// TIA Portal V20 export
FUNCTION "04 T10 LANT Transitions" : Void   // FC1493, LAD
TITLE = TRANSITIONS
{ S7_Optimized_Access := 'TRUE' }
// stored: AutoNumber false, SetENOAutomatically false
   VAR_TEMP
      Aux_real : Real;
   END_VAR
BEGIN

REGION Network 1: ============ TRANSITIONS ============
END_REGION

REGION Network 2: Transitions - Zone Status
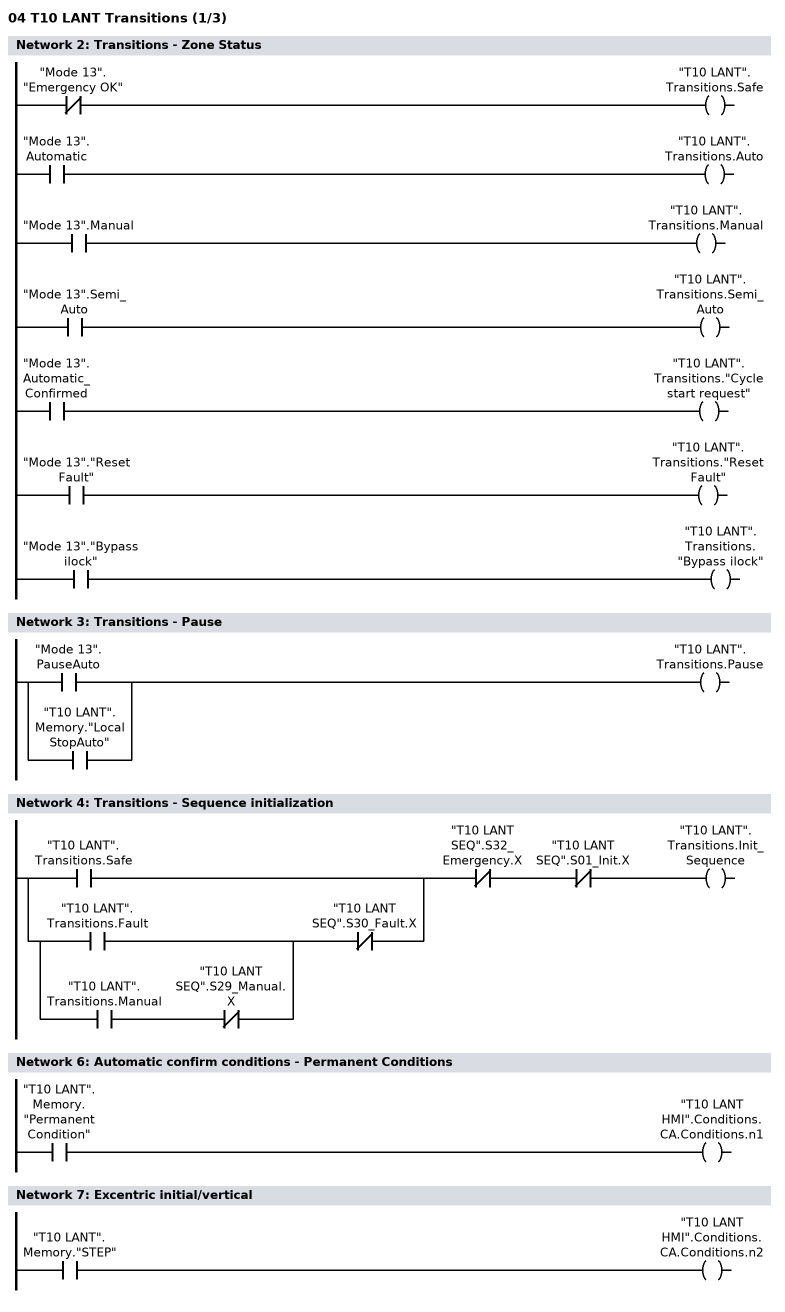
   RUNG wire#powerrail
      I_Contact( "Mode 13"."Emergency OK" )
      Coil( "T10 LANT".Transitions.Safe )
   END_RUNG
   RUNG wire#powerrail
      Contact( "Mode 13".Automatic )
      Coil( "T10 LANT".Transitions.Auto )
   END_RUNG
   RUNG wire#powerrail
      Contact( "Mode 13".Manual )
      Coil( "T10 LANT".Transitions.Manual )
   END_RUNG
   RUNG wire#powerrail
      Contact( "Mode 13".Semi_Auto )
      Coil( "T10 LANT".Transitions.Semi_Auto )
   END_RUNG
   RUNG wire#powerrail
      Contact( "Mode 13".Automatic_Confirmed )
      Coil( "T10 LANT".Transitions."Cycle start request" )
   END_RUNG
   RUNG wire#powerrail
      Contact( "Mode 13"."Reset Fault" )
      Coil( "T10 LANT".Transitions."Reset Fault" )
   END_RUNG
   RUNG wire#powerrail
      Contact( "Mode 13"."Bypass ilock" )
      Coil( "T10 LANT".Transitions."Bypass ilock" )
   END_RUNG
   // the same network as SCL:
   "T10 LANT".Transitions.Safe := NOT "Mode 13"."Emergency OK";
   "T10 LANT".Transitions.Auto := "Mode 13".Automatic;
   "T10 LANT".Transitions.Manual := "Mode 13".Manual;
   "T10 LANT".Transitions.Semi_Auto := "Mode 13".Semi_Auto;
   "T10 LANT".Transitions."Cycle start request" := "Mode 13".Automatic_Confirmed;
   "T10 LANT".Transitions."Reset Fault" := "Mode 13"."Reset Fault";
   "T10 LANT".Transitions."Bypass ilock" := "Mode 13"."Bypass ilock";
END_REGION

REGION Network 3: Transitions - Pause
   RUNG wire#powerrail
      Contact( "Mode 13".PauseAuto )
      wire#w1
      Coil( "T10 LANT".Transitions.Pause )
   END_RUNG
   RUNG wire#powerrail
      Contact( "T10 LANT".Memory."Local StopAuto" )
   END_RUNG wire#w1
   // the same network as SCL:
   "T10 LANT".Transitions.Pause := "Mode 13".PauseAuto OR "T10 LANT".Memory."Local StopAuto";
END_REGION

REGION Network 4: Transitions - Sequence initialization
   RUNG wire#powerrail
      Contact( "T10 LANT".Transitions.Safe )
      wire#w1
      I_Contact( "T10 LANT SEQ".S32_Emergency.X )
      I_Contact( "T10 LANT SEQ".S01_Init.X )
      Coil( "T10 LANT".Transitions.Init_Sequence )
   END_RUNG
   RUNG wire#powerrail
      Contact( "T10 LANT".Transitions.Fault )
      wire#w2
      I_Contact( "T10 LANT SEQ".S30_Fault.X )
   END_RUNG wire#w1
   RUNG wire#powerrail
      Contact( "T10 LANT".Transitions.Manual )
      I_Contact( "T10 LANT SEQ".S29_Manual.X )
   END_RUNG wire#w2
   // the same network as SCL:
   "T10 LANT".Transitions.Init_Sequence := ("T10 LANT".Transitions.Safe OR (("T10 LANT".Transitions.Fault OR ("T10 LANT".Transitions.Manual AND NOT "T10 LANT SEQ".S29_Manual.X)) AND NOT "T10 LANT SEQ".S30_Fault.X)) AND NOT "T10 LANT SEQ".S32_Emergency.X AND NOT "T10 LANT SEQ".S01_Init.X;
END_REGION

REGION Network 5: ============ AUTOMATIC CONFIRM CONDITIONS - 1ST PIECE ============
END_REGION

REGION Network 6: Automatic confirm conditions - Permanent Conditions
   RUNG wire#powerrail
      Contact( "T10 LANT".Memory."Permanent Condition" )
      Coil( "T10 LANT HMI".Conditions.CA.Conditions.n1 )
   END_RUNG
   // the same network as SCL:
   "T10 LANT HMI".Conditions.CA.Conditions.n1 := "T10 LANT".Memory."Permanent Condition";
END_REGION

REGION Network 7: Excentric initial/vertical
   RUNG wire#powerrail
      Contact( "T10 LANT".Memory."STEP" )
      Coil( "T10 LANT HMI".Conditions.CA.Conditions.n2 )
   END_RUNG
   // the same network as SCL:
   "T10 LANT HMI".Conditions.CA.Conditions.n2 := "T10 LANT".Memory."STEP";
END_REGION

REGION Network 8: Transitions - First Piece
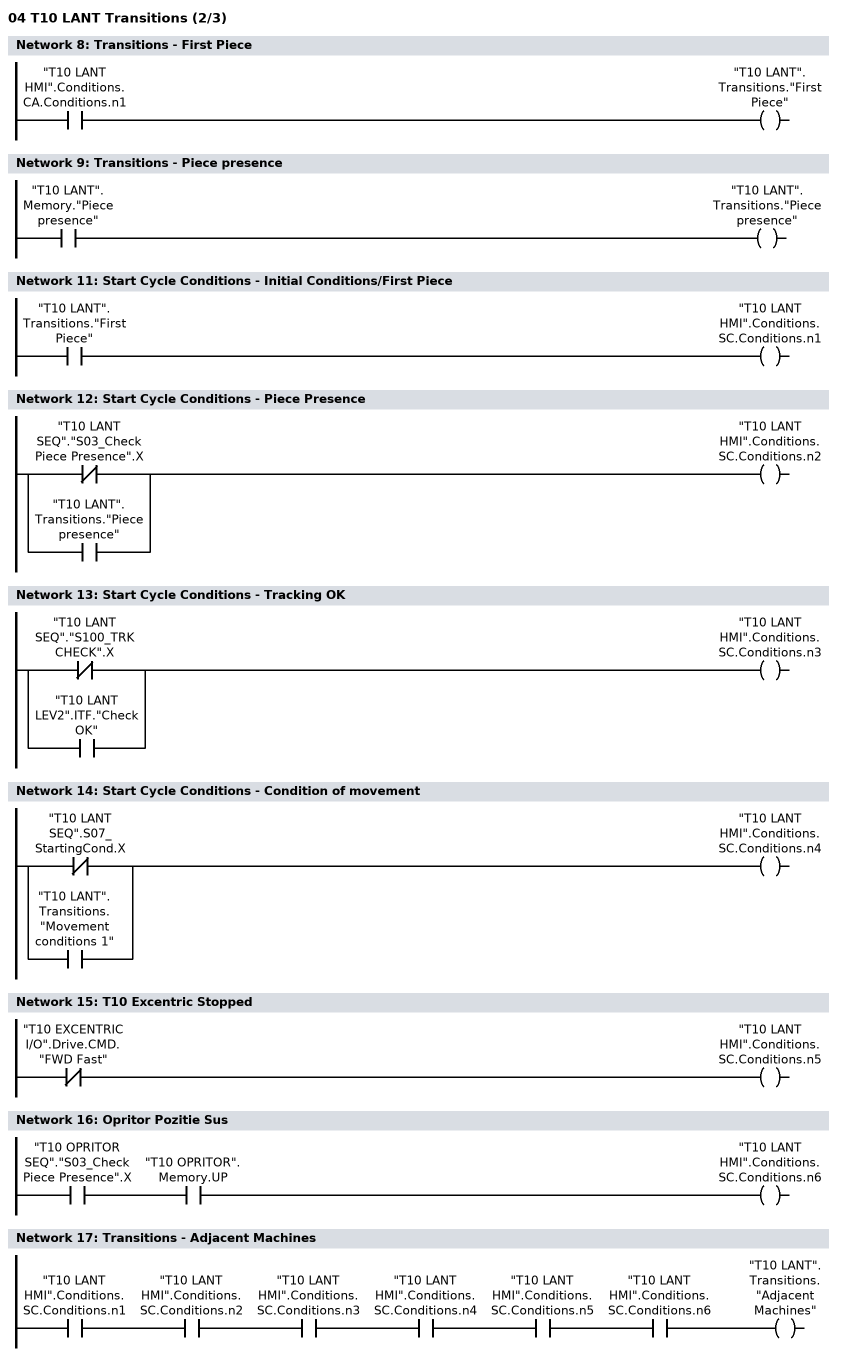
   RUNG wire#powerrail
      Contact( "T10 LANT HMI".Conditions.CA.Conditions.n1 )
      Coil( "T10 LANT".Transitions."First Piece" )
   END_RUNG
   // the same network as SCL:
   "T10 LANT".Transitions."First Piece" := "T10 LANT HMI".Conditions.CA.Conditions.n1;
END_REGION

REGION Network 9: Transitions - Piece presence
   RUNG wire#powerrail
      Contact( "T10 LANT".Memory."Piece presence" )
      Coil( "T10 LANT".Transitions."Piece presence" )
   END_RUNG
   // the same network as SCL:
   "T10 LANT".Transitions."Piece presence" := "T10 LANT".Memory."Piece presence";
END_REGION

REGION Network 10: ============ START CYCLE CONDITIONS ============
END_REGION

REGION Network 11: Start Cycle Conditions - Initial Conditions/First Piece
   RUNG wire#powerrail
      Contact( "T10 LANT".Transitions."First Piece" )
      Coil( "T10 LANT HMI".Conditions.SC.Conditions.n1 )
   END_RUNG
   // the same network as SCL:
   "T10 LANT HMI".Conditions.SC.Conditions.n1 := "T10 LANT".Transitions."First Piece";
END_REGION

REGION Network 12: Start Cycle Conditions - Piece Presence
   RUNG wire#powerrail
      I_Contact( "T10 LANT SEQ"."S03_Check Piece Presence".X )
      wire#w1
      Coil( "T10 LANT HMI".Conditions.SC.Conditions.n2 )
   END_RUNG
   RUNG wire#powerrail
      Contact( "T10 LANT".Transitions."Piece presence" )
   END_RUNG wire#w1
   // the same network as SCL:
   "T10 LANT HMI".Conditions.SC.Conditions.n2 := NOT "T10 LANT SEQ"."S03_Check Piece Presence".X OR "T10 LANT".Transitions."Piece presence";
END_REGION

REGION Network 13: Start Cycle Conditions - Tracking OK
   RUNG wire#powerrail
      I_Contact( "T10 LANT SEQ"."S100_TRK CHECK".X )
      wire#w1
      Coil( "T10 LANT HMI".Conditions.SC.Conditions.n3 )
   END_RUNG
   RUNG wire#powerrail
      Contact( "T10 LANT LEV2".ITF."Check OK" )
   END_RUNG wire#w1
   // the same network as SCL:
   "T10 LANT HMI".Conditions.SC.Conditions.n3 := NOT "T10 LANT SEQ"."S100_TRK CHECK".X OR "T10 LANT LEV2".ITF."Check OK";
END_REGION

REGION Network 14: Start Cycle Conditions - Condition of movement
   RUNG wire#powerrail
      I_Contact( "T10 LANT SEQ".S07_StartingCond.X )
      wire#w1
      Coil( "T10 LANT HMI".Conditions.SC.Conditions.n4 )
   END_RUNG
   RUNG wire#powerrail
      Contact( "T10 LANT".Transitions."Movement conditions 1" )
   END_RUNG wire#w1
   // the same network as SCL:
   "T10 LANT HMI".Conditions.SC.Conditions.n4 := NOT "T10 LANT SEQ".S07_StartingCond.X OR "T10 LANT".Transitions."Movement conditions 1";
END_REGION

REGION Network 15: T10 Excentric Stopped
   RUNG wire#powerrail
      I_Contact( "T10 EXCENTRIC I/O".Drive.CMD."FWD Fast" )
      Coil( "T10 LANT HMI".Conditions.SC.Conditions.n5 )
   END_RUNG
   // the same network as SCL:
   "T10 LANT HMI".Conditions.SC.Conditions.n5 := NOT "T10 EXCENTRIC I/O".Drive.CMD."FWD Fast";
END_REGION

REGION Network 16: Opritor Pozitie Sus
   RUNG wire#powerrail
      Contact( "T10 OPRITOR SEQ"."S03_Check Piece Presence".X )
      Contact( "T10 OPRITOR".Memory.UP )
      Coil( "T10 LANT HMI".Conditions.SC.Conditions.n6 )
   END_RUNG
   // the same network as SCL:
   "T10 LANT HMI".Conditions.SC.Conditions.n6 := "T10 OPRITOR SEQ"."S03_Check Piece Presence".X AND "T10 OPRITOR".Memory.UP;
END_REGION

REGION Network 17: Transitions - Adjacent Machines
   RUNG wire#powerrail
      Contact( "T10 LANT HMI".Conditions.SC.Conditions.n1 )
      Contact( "T10 LANT HMI".Conditions.SC.Conditions.n2 )
      Contact( "T10 LANT HMI".Conditions.SC.Conditions.n3 )
      Contact( "T10 LANT HMI".Conditions.SC.Conditions.n4 )
      Contact( "T10 LANT HMI".Conditions.SC.Conditions.n5 )
      Contact( "T10 LANT HMI".Conditions.SC.Conditions.n6 )
      Coil( "T10 LANT".Transitions."Adjacent Machines" )
   END_RUNG
   // the same network as SCL:
   "T10 LANT".Transitions."Adjacent Machines" := "T10 LANT HMI".Conditions.SC.Conditions.n1 AND "T10 LANT HMI".Conditions.SC.Conditions.n2 AND "T10 LANT HMI".Conditions.SC.Conditions.n3 AND "T10 LANT HMI".Conditions.SC.Conditions.n4 AND "T10 LANT HMI".Conditions.SC.Conditions.n5 AND "T10 LANT HMI".Conditions.SC.Conditions.n6;
END_REGION

REGION Network 18: Pozitia 'Initial'
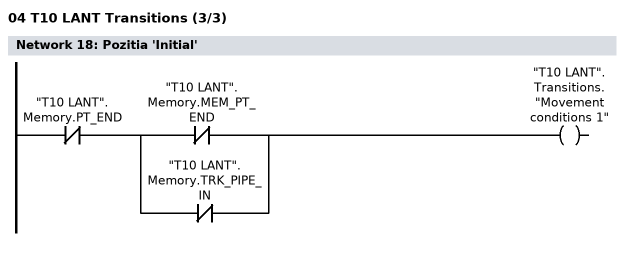
   RUNG wire#powerrail
      I_Contact( "T10 LANT".Memory.PT_END )
      wire#w1
      I_Contact( "T10 LANT".Memory.MEM_PT_END )
      wire#w2
      Coil( "T10 LANT".Transitions."Movement conditions 1" )
   END_RUNG
   RUNG wire#w1
      I_Contact( "T10 LANT".Memory.TRK_PIPE_IN )
   END_RUNG wire#w2
   // the same network as SCL:
   "T10 LANT".Transitions."Movement conditions 1" := NOT "T10 LANT".Memory.PT_END AND (NOT "T10 LANT".Memory.MEM_PT_END OR NOT "T10 LANT".Memory.TRK_PIPE_IN);
END_REGION
END_FUNCTION
